FUNCTION_BLOCK "FB_AxisCtrl"
{ S7_Optimized_Access := 'TRUE' }
VERSION : 2.1
// =====================================================================
// SCARA ABCDE - Axis / Kinematics Control  (Phase 3, 2026-05-21)
//
// The single Motion Control owner. Belongs to the 600 axis/kinematics
// layer; runs in OB30 (CyclicInterrupt_10ms, 10 ms), decoupled from the
// 500 process logic in OB1. All I/O is the consolidated
// GDB_AxisCtrl.LKinCtrl interface (the OB1<->OB30 shared-DB bridge).
//
// V2.1 - adds the kinematic linear-move owner (REGION MoveLinear). The
// auto FBs no longer call MC themselves: they write a target pose into
// GDB_AxisCtrl.LKinCtrl.input.movelinear, hold bo_execute, and read
// output.movelinear.bo_done back. This FB runs the one
// MC_MoveLinearAbsolute on ScaraArm3D - the Huashili motion/process split.
//
// V2.0 - rebuilt on the approved LKinCtrl library (郑老板 approval):
//   - Power:  4x raw MC_Power  ->  1x LKinCtrl_MC_GroupPower
//   - Reset:  5x raw MC_Reset  ->  1x LKinCtrl_MC_GroupReset
//   - Home:   moved OUT to the new FB_Init (LKinCtrl_MC_GroupHome);
//             FB_AxisCtrl only reads back output.bo_homed.
//   - SetTool: kept - MC_SetTool one-shot (Tool[1], the UserFault fix).
//
// Group-level enable for now; per-axis-enable (review 4.2,
// GDB_AxisCtrl.TOCtrl[1..4]) is a follow-on refinement.
// =====================================================================
   VAR
      instGroupPower : "LKinCtrl_MC_GroupPower";
      instGroupReset : "LKinCtrl_MC_GroupReset";
      instMC_SetTool {InstructionName := 'MC_SETTOOL'; LibVersion := '9.0'} : MC_SETTOOL;
      instMoveLinAbs {InstructionName := 'MC_MOVELINEARABSOLUTE'; LibVersion := '9.0'; S7_SetPoint := 'False'} : MC_MOVELINEARABSOLUTE;
      statToolActivated : Bool;   // one-shot SetTool latch; cleared by memory reset
   END_VAR

   VAR_TEMP
      tempPos : Array[1..6] of LReal;   // Cartesian Position array for MC_MoveLinearAbsolute
   END_VAR


BEGIN

    REGION Power
        // Enable all kinematic axes via the library group-power FB.
        // startMode / stopMode arrays come from the consolidated config.
        #instGroupPower(enable    := "GDB_AxisCtrl".LKinCtrl.input.bo_enable,
                        startMode := "GDB_AxisCtrl".LKinCtrl.input.configuration.power.startMode,
                        stopMode  := "GDB_AxisCtrl".LKinCtrl.input.configuration.power.stopMode,
                        axesGroup := "ScaraArm3D");
        "GDB_AxisCtrl".LKinCtrl.output.bo_enabled := #instGroupPower.axesEnabled;
    END_REGION

    REGION Reset
        // Reset all axes + the kinematics TO via the library group-reset FB.
        #instGroupReset(execute   := "GDB_AxisCtrl".LKinCtrl.input.bo_reset,
                        restart   := "GDB_AxisCtrl".LKinCtrl.input.configuration.reset.restart,
                        axesGroup := "ScaraArm3D");
    END_REGION

    REGION Fault
        "GDB_AxisCtrl".LKinCtrl.output.bo_fault := #instGroupPower.error
                                                   OR #instGroupReset.error;
    END_REGION

    REGION SetTool
        // One-shot Tool[1] activation once the group is enabled. Without an
        // active tool, MC_MoveLinearAbsolute returns UserFault (documented
        // root cause). Idempotent: latches statToolActivated, drops Execute
        // after Done. Cleared by memory reset.
        IF "GDB_AxisCtrl".LKinCtrl.output.bo_enabled AND NOT #statToolActivated THEN
            #instMC_SetTool(AxesGroup  := "ScaraArm3D",
                            Execute    := TRUE,
                            ToolNumber := 1);
            IF #instMC_SetTool.Done THEN
                #instMC_SetTool(AxesGroup := "ScaraArm3D",
                                Execute   := FALSE);
                #statToolActivated := TRUE;
            END_IF;
        END_IF;
    END_REGION

    REGION MoveLinear
        // Kinematic linear move on ScaraArm3D. The auto FBs (OB1) write the
        // target pose + dynamics into GDB_AxisCtrl.LKinCtrl.input.movelinear
        // and hold bo_execute; this region runs the one MC_MoveLinearAbsolute
        // and mirrors its status into output.movelinear for the auto FB's
        // wait-in-place step. BufferMode 1 (buffered) - the auto CASE
        // serializes moves (one per step, waits for Done), so no
        // cross-command blending is needed.
        #tempPos[1] := "GDB_AxisCtrl".LKinCtrl.input.movelinear.targetposition.x;
        #tempPos[2] := "GDB_AxisCtrl".LKinCtrl.input.movelinear.targetposition.y;
        #tempPos[3] := "GDB_AxisCtrl".LKinCtrl.input.movelinear.targetposition.z;
        #tempPos[4] := "GDB_AxisCtrl".LKinCtrl.input.movelinear.targetposition.a;
        #tempPos[5] := "GDB_AxisCtrl".LKinCtrl.input.movelinear.targetposition.b;
        #tempPos[6] := "GDB_AxisCtrl".LKinCtrl.input.movelinear.targetposition.c;

        #instMoveLinAbs(AxesGroup    := "ScaraArm3D",
                        Execute      := "GDB_AxisCtrl".LKinCtrl.input.movelinear.bo_execute,
                        Position     := #tempPos,
                        Velocity     := "GDB_AxisCtrl".LKinCtrl.input.movelinear.r64_velocity,
                        Acceleration := "GDB_AxisCtrl".LKinCtrl.input.movelinear.r64_acceleration,
                        Deceleration := "GDB_AxisCtrl".LKinCtrl.input.movelinear.r64_deceleration,
                        Jerk         := "GDB_AxisCtrl".LKinCtrl.input.movelinear.r64_jerk,
                        BufferMode   := 1);

        "GDB_AxisCtrl".LKinCtrl.output.movelinear.bo_done           := #instMoveLinAbs.Done;
        "GDB_AxisCtrl".LKinCtrl.output.movelinear.bo_busy           := #instMoveLinAbs.Busy;
        "GDB_AxisCtrl".LKinCtrl.output.movelinear.bo_active         := #instMoveLinAbs.Active;
        "GDB_AxisCtrl".LKinCtrl.output.movelinear.bo_error          := #instMoveLinAbs.Error;
        "GDB_AxisCtrl".LKinCtrl.output.movelinear.bo_commandaborted := #instMoveLinAbs.CommandAborted;
    END_REGION

    REGION StatusDerived
        // bo_ready = enabled AND homed AND NOT fault. bo_homed is written
        // by FB_Init - call FB_Init before FB_AxisCtrl in OB30.
        "GDB_AxisCtrl".LKinCtrl.output.bo_ready :=
            "GDB_AxisCtrl".LKinCtrl.output.bo_enabled
            AND "GDB_AxisCtrl".LKinCtrl.output.bo_homed
            AND NOT "GDB_AxisCtrl".LKinCtrl.output.bo_fault;
    END_REGION

END_FUNCTION_BLOCK
